FUNCTION_BLOCK E_Merge16 (* Composite Function Block Type *)
  (* Standard: 61499-2 *)
  (* Version 0.0, 2018-12-21, 4DIAC-IDE, 4DIAC-Consortium *)
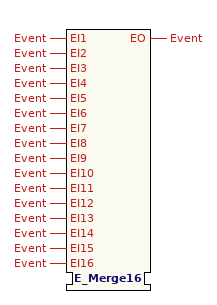
  EVENT_INPUT
    EI1; (* Initialization Request *)
    EI2;
    EI3;
    EI4;
    EI5;
    EI6;
    EI7;
    EI8;
    EI9;
    EI10;
    EI11;
    EI12;
    EI13;
    EI14;
    EI15;
    EI16;
  END_EVENT
  EVENT_OUTPUT
    EO; (* Initialization Confirm *)
  END_EVENT
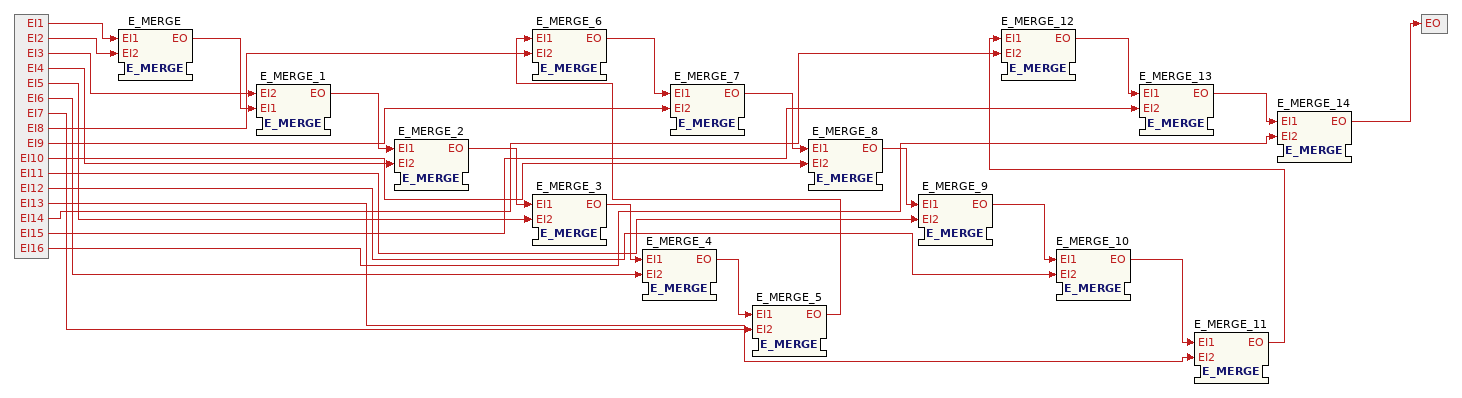
  FBS
    E_MERGE : E_MERGE;
    E_MERGE_1 : E_MERGE;
    E_MERGE_2 : E_MERGE;
    E_MERGE_3 : E_MERGE;
    E_MERGE_4 : E_MERGE;
    E_MERGE_5 : E_MERGE;
    E_MERGE_6 : E_MERGE;
    E_MERGE_7 : E_MERGE;
    E_MERGE_8 : E_MERGE;
    E_MERGE_9 : E_MERGE;
    E_MERGE_10 : E_MERGE;
    E_MERGE_11 : E_MERGE;
    E_MERGE_12 : E_MERGE;
    E_MERGE_13 : E_MERGE;
    E_MERGE_14 : E_MERGE;
  END_FBS
  EVENT_CONNECTIONS
    EI1 TO E_MERGE.EI1;
    EI2 TO E_MERGE.EI2;
    EI3 TO E_MERGE_1.EI2;
    E_MERGE.EO TO E_MERGE_1.EI1;
    E_MERGE_1.EO TO E_MERGE_2.EI1;
    EI4 TO E_MERGE_2.EI2;
    E_MERGE_2.EO TO E_MERGE_3.EI1;
    EI5 TO E_MERGE_3.EI2;
    E_MERGE_3.EO TO E_MERGE_4.EI1;
    EI6 TO E_MERGE_4.EI2;
    E_MERGE_4.EO TO E_MERGE_5.EI1;
    EI7 TO E_MERGE_5.EI2;
    E_MERGE_5.EO TO E_MERGE_6.EI1;
    EI8 TO E_MERGE_6.EI2;
    E_MERGE_6.EO TO E_MERGE_7.EI1;
    EI9 TO E_MERGE_7.EI2;
    E_MERGE_7.EO TO E_MERGE_8.EI1;
    EI10 TO E_MERGE_8.EI2;
    E_MERGE_8.EO TO E_MERGE_9.EI1;
    EI11 TO E_MERGE_9.EI2;
    E_MERGE_9.EO TO E_MERGE_10.EI1;
    EI12 TO E_MERGE_10.EI2;
    E_MERGE_10.EO TO E_MERGE_11.EI1;
    EI13 TO E_MERGE_11.EI2;
    E_MERGE_11.EO TO E_MERGE_12.EI1;
    EI14 TO E_MERGE_12.EI2;
    E_MERGE_12.EO TO E_MERGE_13.EI1;
    EI15 TO E_MERGE_13.EI2;
    E_MERGE_13.EO TO E_MERGE_14.EI1;
    EI16 TO E_MERGE_14.EI2;
    E_MERGE_14.EO TO EO;
  END_CONNECTIONS
END_FUNCTION_BLOCK
